// SIMATIC STEP 7 (V5.x) project PROJEKT_L
// CPU: CPU 315-2 DP
// station: P_ADR_BUS
// station: Hardware
// station: SIMATIC 300(1)
// station: Configuration
// station: P_ADR_BUS
// program: S7 Program(1)
// program: MICROMASTER_420

SYMBOL_TABLE
"FOR_READ"	DB 1	DB 1
"FOR_W"	DB 2	DB 2
"DB3"	DB 3	DB 3
"set bit and allarms"	DB 4	DB 4
"GET"	FB 14	FB 14	// Read Data From a Remote CPU
"POS_INIT"	FC 0	FC 0	// Initialize channel datablock
"Micromaster config"	FC 1	FC 1
"POS_MSRM"	FC 3	FC 3	// Measurement Values
"GT_DT"	FC 14	FC 14	// Greater Than DT
"Always on"	M 0.1	BOOL
"always off"	M 0.2	BOOL
"are"	M 0.4	BOOL
"1"	M 0.5	BOOL
"inter look"	M 0.6	BOOL
"revers"	M 0.7	BOOL
"ack"	M 1.0	BOOL
"Main block"	OB 1	OB 1
"DPRD_DAT"	SFC 14	SFC 14	// Read Consistent Data of a Standard DP Slave
"DPWR_DAT"	SFC 15	SFC 15	// Write Consistent Data to a Standard DP Slave
"RD_REC"	SFC 59	SFC 59	// Read a Data Record
END_SYMBOL_TABLE

// FB 14: know-how protected block, not included

// FC 0: know-how protected block, not included

FUNCTION "Micromaster config" : VOID	// FC 1
TITLE = Micromaster configuration function
VERSION : 0.1
VAR_TEMP
  TEMPD1 : DINT ;
  TEMPR2 : REAL ;
  TEMPR3 : REAL ;
  TEMPR73 : REAL ;
END_VAR
BEGIN
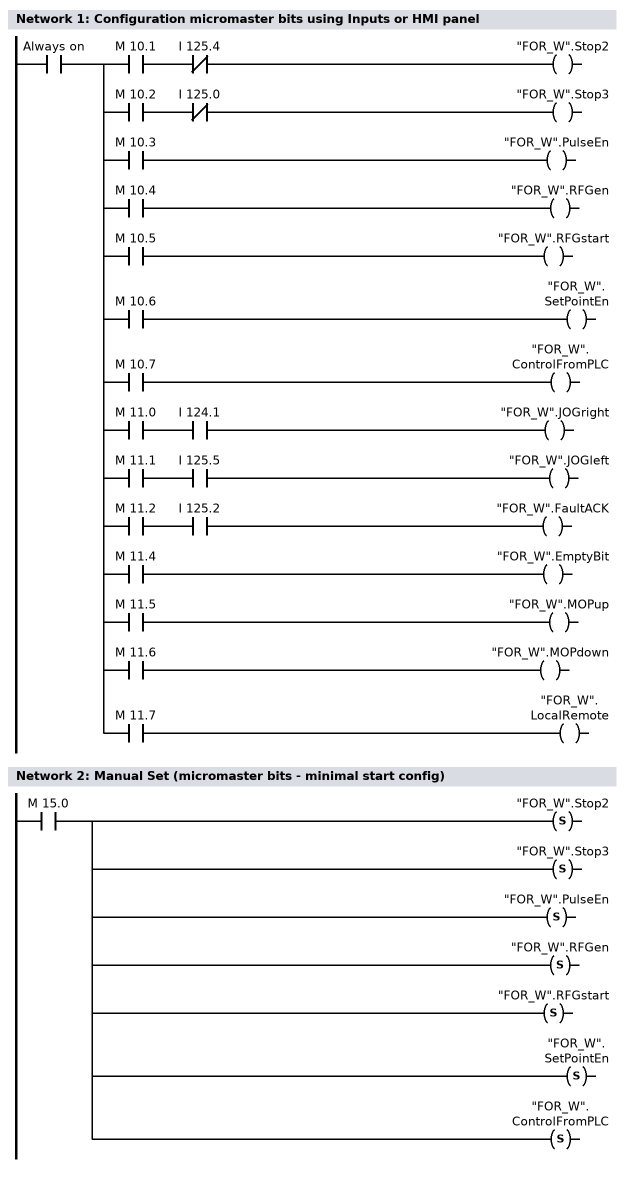
NETWORK
TITLE = Configuration micromaster bits using Inputs or HMI panel 
      A     "Always on";
      =     L 16.0;
      A     L 16.0;
      A     M 10.1;
      AN    I 125.4;
      =     "FOR_W".Stop2;
      A     L 16.0;
      A     M 10.2;
      AN    I 125.0;
      =     "FOR_W".Stop3;
      A     L 16.0;
      A     M 10.3;
      =     "FOR_W".PulseEn;
      A     L 16.0;
      A     M 10.4;
      =     "FOR_W".RFGen;
      A     L 16.0;
      A     M 10.5;
      =     "FOR_W".RFGstart;
      A     L 16.0;
      A     M 10.6;
      =     "FOR_W".SetPointEn;
      A     L 16.0;
      A     M 10.7;
      =     "FOR_W".ControlFromPLC;
      A     L 16.0;
      A     M 11.0;
      A     I 124.1;
      =     "FOR_W".JOGright;
      A     L 16.0;
      A     M 11.1;
      A     I 125.5;
      =     "FOR_W".JOGleft;
      A     L 16.0;
      A     M 11.2;
      A     I 125.2;
      =     "FOR_W".FaultACK;
      A     L 16.0;
      A     M 11.4;
      =     "FOR_W".EmptyBit;
      A     L 16.0;
      A     M 11.5;
      =     "FOR_W".MOPup;
      A     L 16.0;
      A     M 11.6;
      =     "FOR_W".MOPdown;
      A     L 16.0;
      A     M 11.7;
      =     "FOR_W".LocalRemote;
NETWORK
TITLE = Manual Set (micromaster bits - minimal start config)
      A     M 15.0;
      S     "FOR_W".Stop2;
      S     "FOR_W".Stop3;
      S     "FOR_W".PulseEn;
      S     "FOR_W".RFGen;
      S     "FOR_W".RFGstart;
      S     "FOR_W".SetPointEn;
      S     "FOR_W".ControlFromPLC;
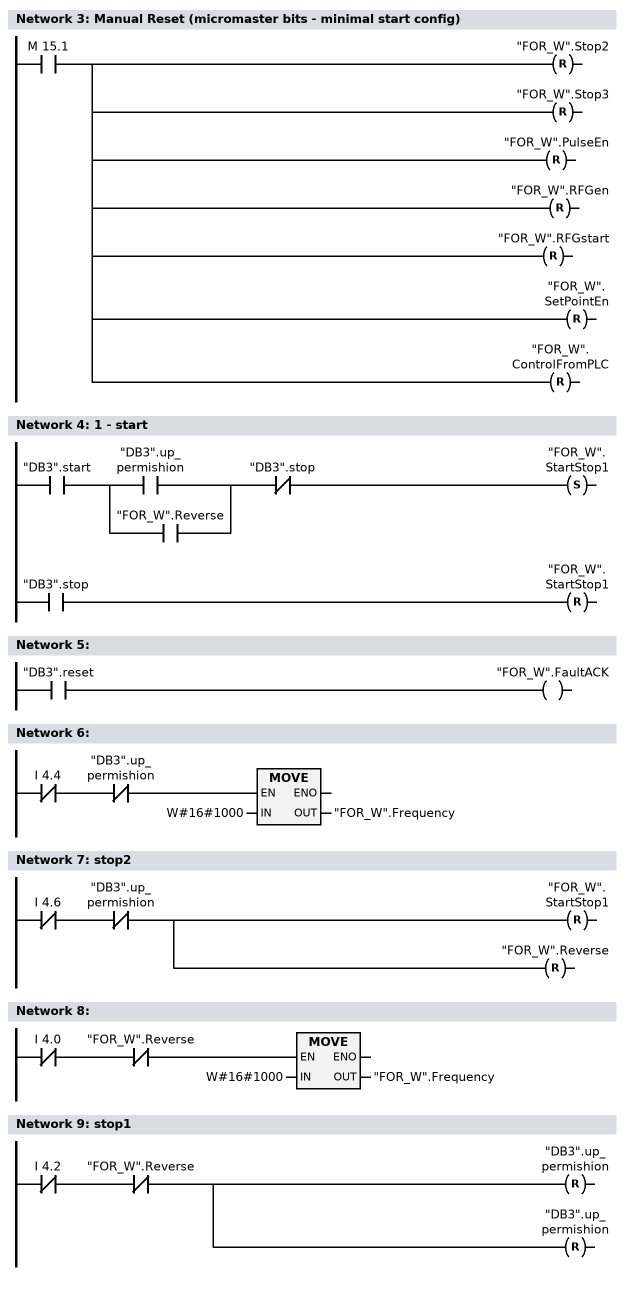
NETWORK
TITLE = Manual Reset (micromaster bits - minimal start config)
      A     M 15.1;
      R     "FOR_W".Stop2;
      R     "FOR_W".Stop3;
      R     "FOR_W".PulseEn;
      R     "FOR_W".RFGen;
      R     "FOR_W".RFGstart;
      R     "FOR_W".SetPointEn;
      R     "FOR_W".ControlFromPLC;
NETWORK
TITLE = 1 - start 
      A     "DB3".start;
      A(;
      O     "DB3".up_permishion;
      O     "FOR_W".Reverse;
      );
      AN    "DB3".stop;
      S     "FOR_W".StartStop1;
      A     "DB3".stop;
      R     "FOR_W".StartStop1;
      NOP   0;
NETWORK
TITLE =
      A     "DB3".reset;
      =     "FOR_W".FaultACK;
NETWORK
TITLE =
      AN    I 4.4;
      AN    "DB3".up_permishion;
      JNB   _001;
      L     W#16#1000;
      T     "FOR_W".Frequency;
_001: NOP   0;
NETWORK
TITLE = stop2
      AN    I 4.6;
      AN    "DB3".up_permishion;
      R     "FOR_W".StartStop1;
      R     "FOR_W".Reverse;
NETWORK
TITLE =
      AN    I 4.0;
      AN    "FOR_W".Reverse;
      JNB   _002;
      L     W#16#1000;
      T     "FOR_W".Frequency;
_002: NOP   0;
NETWORK
TITLE = stop1
      AN    I 4.2;
      AN    "FOR_W".Reverse;
      R     "DB3".up_permishion;
      R     "DB3".up_permishion;
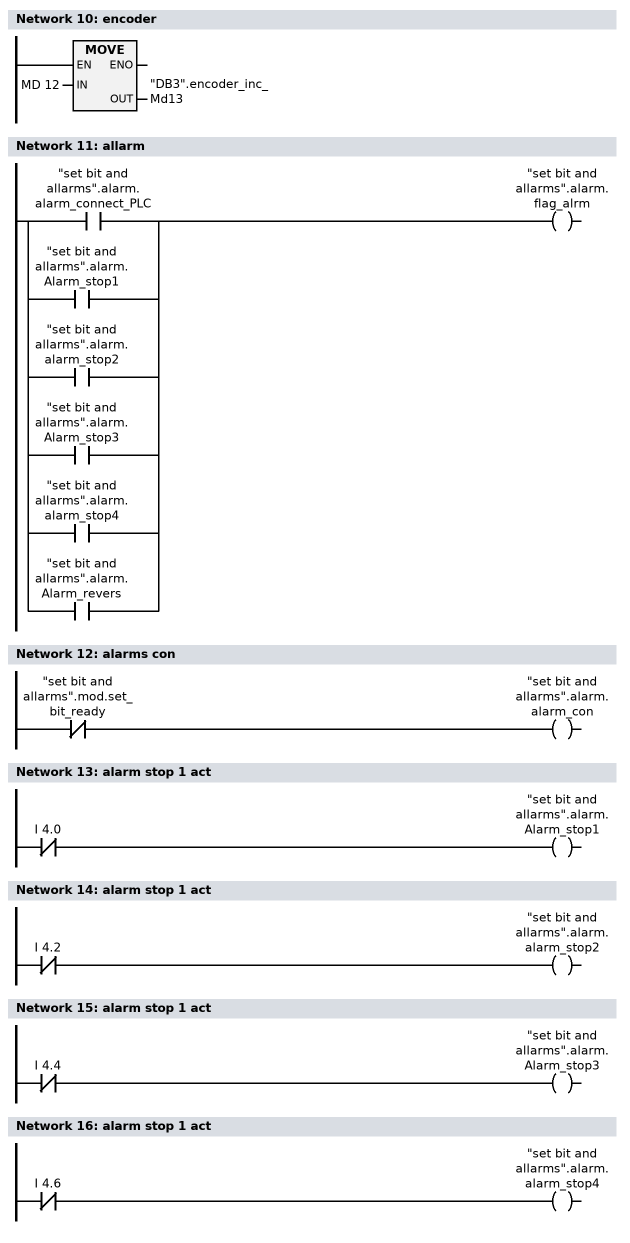
NETWORK
TITLE = encoder
      L     MD 12;
      T     "DB3".encoder_inc_Md13;
      NOP   0;
NETWORK
TITLE = allarm
      O     "set bit and allarms".alarm.alarm_connect_PLC;
      O     "set bit and allarms".alarm.Alarm_stop1;
      O     "set bit and allarms".alarm.alarm_stop2;
      O     "set bit and allarms".alarm.Alarm_stop3;
      O     "set bit and allarms".alarm.alarm_stop4;
      O     "set bit and allarms".alarm.Alarm_revers;
      =     "set bit and allarms".alarm.flag_alrm;
NETWORK
TITLE = alarms con 
      AN    "set bit and allarms".mod.set_bit_ready;
      =     "set bit and allarms".alarm.alarm_con;
NETWORK
TITLE = alarm stop 1 act
      AN    I 4.0;
      =     "set bit and allarms".alarm.Alarm_stop1;
NETWORK
TITLE = alarm stop 1 act
      AN    I 4.2;
      =     "set bit and allarms".alarm.alarm_stop2;
NETWORK
TITLE = alarm stop 1 act
      AN    I 4.4;
      =     "set bit and allarms".alarm.Alarm_stop3;
NETWORK
TITLE = alarm stop 1 act
      AN    I 4.6;
      =     "set bit and allarms".alarm.alarm_stop4;
END_FUNCTION

FUNCTION FC 2 : VOID
VERSION : 0.1
BEGIN
// (block stored without names or comments; labels and parameter names are numbered)
END_FUNCTION

// FC 3: know-how protected block, not included

// FC 14: know-how protected block, not included

DATA_BLOCK "FOR_READ"	// DB 1
VERSION : 0.1
  STRUCT
   ValueReached : BOOL ;	//Set frequency reached
   PZDcontrol : BOOL ;	//Control priority (1 - master control)
   MaximumReached : BOOL ;	//Maximum frequency reached
   MotorCurLim : BOOL ;	//Warning: Motor current limit
   MotorHoldBrake : BOOL ;	//Motor holding brake
   MotorOverload : BOOL ;	//Motor overload
   MotorRunsDir : BOOL ;	//Motor runs direction (1 - right 0 - left)
   InverterOverl : BOOL ;	//Inverter overload
   DriveReady : BOOL ;	//Drive ready
   DriveReadyRun : BOOL ;	//Drive ready to run
   DriveRunning : BOOL ;	//Drive running
   DriveFaultAct : BOOL ;	//Drive fault
   Stop2Act : BOOL ;	//Stop2 active
   Stop3Act : BOOL ;	//Stop3 active
   ONinhibitAct : BOOL ;	//Launch locked
   DriveWarAct : BOOL ;	//Drive warning
   Frequency : INT  := 10;	//Current frequency
  END_STRUCT ;	
BEGIN
   Frequency := 10;
END_DATA_BLOCK

DATA_BLOCK "FOR_W"	// DB 2
VERSION : 0.1
  STRUCT
   JOGright : BOOL ;	//slow scroll rigth (+5 Hz)
   JOGleft : BOOL ;	//slow scroll left (-5 Hz)
   ControlFromPLC : BOOL ;	//enable control from PLC
   Reverse : BOOL ;	//1 - left scroll 0 - right scroll
   EmptyBit : BOOL ;	//not used
   MOPup : BOOL ;	//motor potentiometer MOP up
   MOPdown : BOOL ;	//motor potentiometer MOP down
   LocalRemote : BOOL ;	//not used
   StartStop1 : BOOL ;	//1 - start 0 - middle stop
   Stop2 : BOOL ;	//stop without brake
   Stop3 : BOOL ;	//fast stop
   PulseEn : BOOL ;	//inverter pulse enable
   RFGen : BOOL ;	//RFG (intensity control) enable
   RFGstart : BOOL ;	//RFG (intensity control)start
   SetPointEn : BOOL ;	//set point enable
   FaultACK : BOOL ;	//fault acknowledge
   Frequency : WORD ;	//set frequency
  END_STRUCT ;	
BEGIN
END_DATA_BLOCK

DATA_BLOCK "DB3"	// DB 3
VERSION : 0.1
  STRUCT
   Frequency_int : INT ;	//Frequency as integer
   Frequency_word : WORD ;	//Frequency as word
   reset : BOOL ;
   con_for_reset : BOOL ;
   permision_for_start : BOOL ;
   encoder_inc_Md13 : WORD ;
   start : BOOL ;
   stop : BOOL ;
   up_permishion : BOOL ;
   animati_permishion : BOOL ;
  END_STRUCT ;	
BEGIN
END_DATA_BLOCK

DATA_BLOCK "set bit and allarms"	// DB 4
VERSION : 0.1
  STRUCT
   alarm : STRUCT
    flag_alrm : BOOL ;
    alarm_connect_PLC : BOOL ;
    Alarm_stop1 : BOOL  := TRUE;
    alarm_stop2 : BOOL ;
    Alarm_stop3 : BOOL ;
    alarm_stop4 : BOOL ;
    Alarm_revers : BOOL ;
    alarm_con : BOOL ;
   END_STRUCT ;
   mod : STRUCT
    mod_enc_1c : BOOL ;
    mod_set_frec_1C : BOOL ;
    flag_mod_enc : BOOL ;
    flag_mod_fc : BOOL ;
    set_bit_ready : BOOL ;
    reset_bit_ready : BOOL ;
   END_STRUCT ;
  END_STRUCT ;	
BEGIN
END_DATA_BLOCK

ORGANIZATION_BLOCK "Main block"	// OB 1
TITLE = "Main Program Sweep (Cycle)"
VERSION : 0.1
VAR_TEMP
  OB1_EV_CLASS : BYTE ;	//Bits 0-3 = 1 (Coming event), Bits 4-7 = 1 (Event class 1)
  OB1_SCAN_1 : BYTE ;	//1 (Cold restart scan 1 of OB 1), 3 (Scan 2-n of OB 1)
  OB1_PRIORITY : BYTE ;	//Priority of OB Execution
  OB1_OB_NUMBR : BYTE ;	//1 (Organization block 1, OB1)
  OB1_RESERVED_1 : BYTE ;	//Reserved for system
  OB1_RESERVED_2 : BYTE ;	//Reserved for system
  OB1_PREV_CYCLE : INT ;	//Cycle time of previous OB1 scan (milliseconds)
  OB1_MIN_CYCLE : INT ;	//Minimum cycle time of OB1 (milliseconds)
  OB1_MAX_CYCLE : INT ;	//Maximum cycle time of OB1 (milliseconds)
  OB1_DATE_TIME : DATE_AND_TIME ;	//Date and time OB1 started
END_VAR
BEGIN
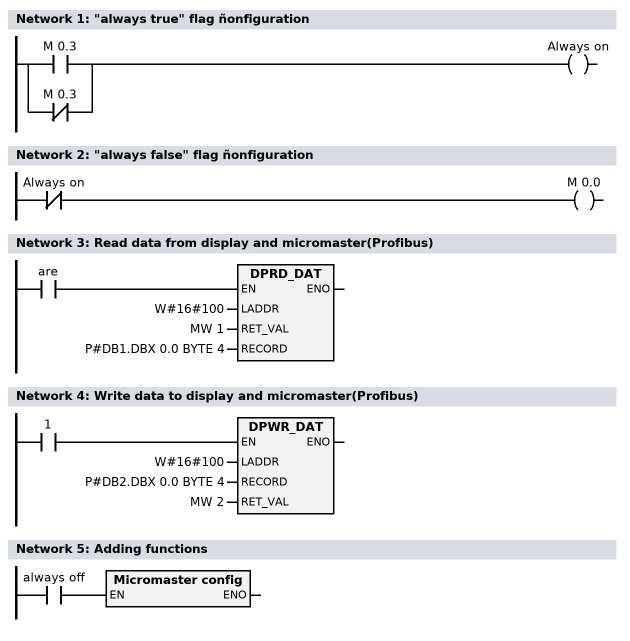
NETWORK
TITLE = "always true" flag ñonfiguration 
      O     M 0.3;
      ON    M 0.3;
      =     "Always on";
NETWORK
TITLE = "always false" flag ñonfiguration 
      AN    "Always on";
      =     M 0.0;
NETWORK
TITLE = Read data from display and micromaster(Profibus)
      A     "are";
      JNB   _001;
      CALL  "DPRD_DAT" (
           LADDR                    := W#16#100,
           RET_VAL                  := MW 1,
           RECORD                   := P#DB1.DBX 0.0 BYTE 4);
_001: NOP   0;
NETWORK
TITLE = Write data to display and micromaster(Profibus)
      A     "1";
      JNB   _002;
      CALL  "DPWR_DAT" (
           LADDR                    := W#16#100,
           RECORD                   := P#DB2.DBX 0.0 BYTE 4,
           RET_VAL                  := MW 2);
_002: NOP   0;
NETWORK
TITLE = Adding functions
      A     "always off";
      JNB   _003;
      CALL  "Micromaster config";
_003: NOP   0;
END_ORGANIZATION_BLOCK

DATA_BLOCK DB 1200
VERSION : 0.0
BEGIN
// 248 bytes; values not shown
END_DATA_BLOCK
